# EPICS alarm handler configuration: mps_database/bare/alarms/areas/mpln_sltd_mp01.alhConfig
GROUP NULL MPLN:SLTD:MP01:1
$ALIAS MPS Link Node 96
$GUIDANCE
LTUH MPS
   Group Name: MPLN:SLTD:MP01:1
   Summary PV:  MPLN:SLTD:MP01:1:STATSUMY
$END
CHANNEL  MPLN:SLTD:MP01:1    MPLN:SLTD:MP01:1:MPS_EN_RBV		-----
CHANNEL  MPLN:SLTD:MP01:1    MPLN:SLTD:MP01:1:LC1_MODE_RBV		-----
